// TIA Portal V17 export
// export: Created 2022-02-03T14:45:17.0730738Z, ExportSetting WithDefaults, DisplayName Totally Integrated Automation Portal, DisplayVersion V17, DisplayName TIA Portal Openness, DisplayVersion V17, DisplayName TIA Portal Version Control Interface, DisplayVersion V17, DisplayName SINAMICS Startdrive Advanced, DisplayVersion V17, DisplayName SINAMICS Startdrive G130, G150, S120, S150, SINAMICS MV, S210, DisplayVersion V17, DisplayName SINAMICS Startdrive G110M, G120, G120C, G120D, G120P, G115D, DisplayVersion V17, DisplayName STEP 7 Professional, DisplayVersion V17, DisplayName STEP 7 Safety, DisplayVersion V17, DisplayName WinCC Advanced, DisplayVersion V17
TYPE "typeConveyorInput"
// stored: Access Published, IsFailsafeCompliant false
   STRUCT
      B_lightBarrier : Bool;
      S_bay1 : Bool;
      S_bay2 : Bool;
      S_bay3 : Bool;
      S_lightBarrier : Bool;
      B_bay1 : Bool;
      B_bay2 : Bool;
      B_bay3 : Bool;
   END_STRUCT;
END_TYPE
